// TIA Portal project "PLC_ABB_Drive" (V15)

(* hardware
DEVICE "S7-1200 station_1"  S7-1200 Station
   slot 0: "Rack_0"  S7-1200 Rack  Rack  V1.0
   slot 1: "PLC_1"  CPU 1212C DC/DC/DC  6ES7 212-1AE31-0XB0  V3.0
   slot 101: "CM 1243-5"  CM 1243-5  6GK7 243-5DX30-0XE0  V1.3
DEVICE "GSD device_1"  GSD.Device
   slot 0: "Slave_1"  6SE640X-1PB00-0AA0  V1.0
   slot 0: "Rack_0"  Rail
*)

// ===== PLC "PLC_1"  CPU 1212C DC/DC/DC =====

VAR_GLOBAL   // PLC tag table "Default tag table"
   "Tag_1" AT %ID260 : DWord;
   "Tag_2" AT %MW100 : Word;
   "InicioVariador" AT %M0.0 : Bool;
   "Tag_3" AT %M0.1 : Bool;
   "Tag_4" AT %M0.2 : Bool;
   "Tag_5" AT %M0.3 : Bool;
   "Tag_6" AT %M0.4 : Bool;
   "Tag_7" AT %M0.5 : Bool;
   "Tag_8" AT %M0.6 : Bool;
   "Tag_9" AT %M0.7 : Bool;
   "Tag_10" AT %M1.0 : Bool;
   "Tag_11" AT %M1.1 : Bool;
   "Tag_12" AT %M1.2 : Bool;
   "Tag_13" AT %M1.4 : Bool;
   "Tag_14" AT %M1.3 : Bool;
   "Tag_15" AT %M1.5 : Bool;
   "Tag_16" AT %M1.6 : Bool;
   "Tag_17" AT %M1.7 : Bool;
   "Tag_18" AT %M2.0 : Bool;
   "LeerValorParam" AT %ID260 : DWord;
   "Tag_20" AT %QW266 : Word;
   "ParametrosDeControl" AT %QW264 : Word;
   "VelocidadControl" AT %MW90 : Word;
   "ParametroControlVel." AT %QW268 : Int;
   "Tag_21" AT %IW264 : Word;
   "Parametro" AT %QW256 : Word;
   "Indice" AT %QW258 : Int;
   "Tag_24" AT %QW260 : Word;
   "ValorParametro" AT %QD260 : Real;
   "LeerParametro" AT %IW256 : Word;
   "ParamRecibido" AT %MW6 : Word;
   "LeerIndice" AT %IW258 : Int;
   "IndiceRecibido" AT %MW8 : Int;
   "VlrParamRecibido" AT %MD10 : DWord;
END_VAR

TYPE "inn"
   STRUCT
      JogDerecha : Bool;
      JogIzquierda : Bool;
      controlPLC : Bool;
      InversionGiro : Bool;
      libre : Bool;
      potenciometroarriba : Bool;
      potenciometroabajo : Bool;
      "mando-local-remoto" : Bool;
      start : Bool;
      stop : Bool;
      "stop-rapido" : Bool;
      "generador-rampa" : Bool;
      "rampa-on" : Bool;
      "rampa-off" : Bool;
      "rampa-start" : Bool;
      "alarma-fallo" : Bool;
      VelVariador : Int;
   END_STRUCT;
END_TYPE

TYPE "out1"
   STRUCT
      Setpoint_on_off : Bool;
      MasterControlReq : Bool;
      F_reached : Bool;
      Alarm_currentLim : Bool;
      MotorHoldBreake : Bool;
      MotorOverload : Bool;
      CW0_CWW1 : Bool;
      ConverterOverload : Bool;
      ReadyForOn : Bool;
      ReadyToRun : Bool;
      OperationEnable : Bool;
      Fault1 : Bool;
      Off2Command : Bool;
      Off3Command : Bool;
      StartLockout : Bool;
      Alarm : Bool;
      StatusSpeed : Int;
   END_STRUCT;
END_TYPE

DATA_BLOCK "LecturadelVariador"   // DB1
{ S7_Optimized_Access := 'FALSE' }
VERSION : 0.1
   VAR
      estadodelvariador : "out1";
   END_VAR
BEGIN
END_DATA_BLOCK

DATA_BLOCK "ControldelVariador"   // DB2
{ S7_Optimized_Access := 'FALSE' }
VERSION : 0.1
   VAR
      controlvariador : "inn";
   END_VAR
BEGIN
END_DATA_BLOCK

FUNCTION_BLOCK "Block_1"   // FB1, FBD
{ S7_Optimized_Access := 'TRUE' }
VERSION : 0.1
BEGIN
END_FUNCTION_BLOCK

ORGANIZATION_BLOCK "Main"   // OB1, LAD, ProgramCycle
TITLE = "Main Program Sweep (Cycle)"
{ S7_Optimized_Access := 'TRUE' }
VERSION : 0.1
BEGIN

REGION Network 1
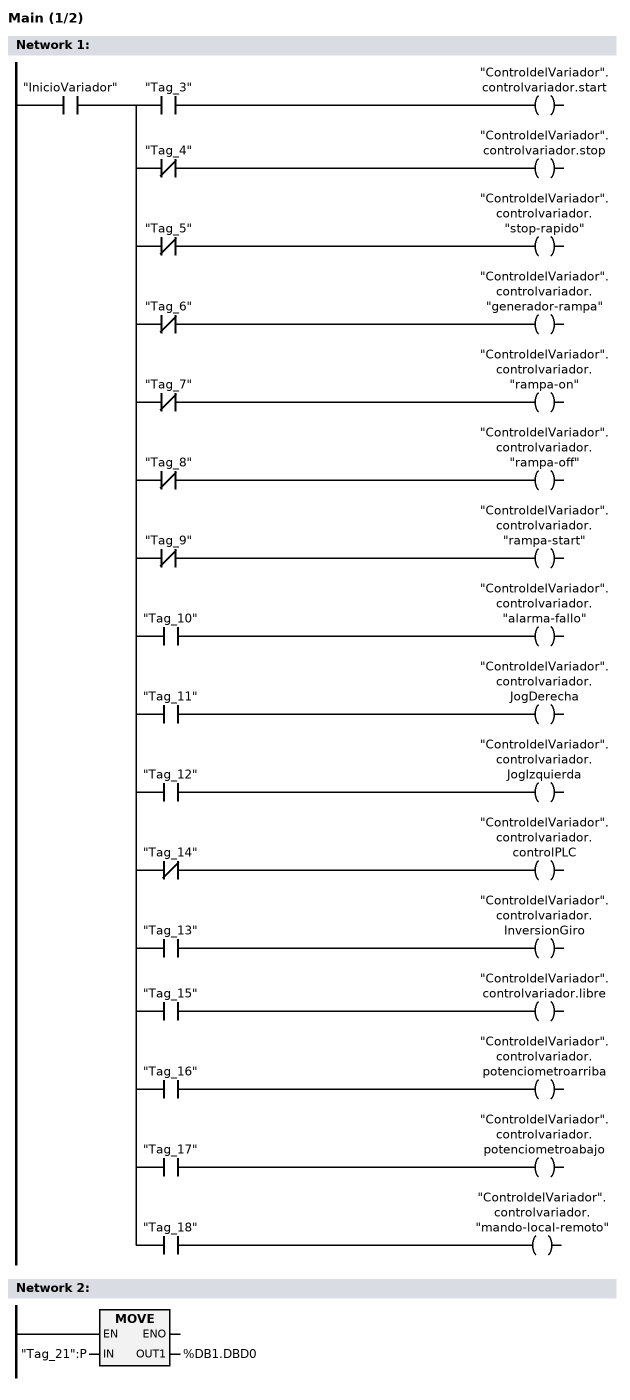
   RUNG wire#powerrail
      Contact( "InicioVariador" )
      wire#w1
      Contact( "Tag_3" )
      Coil( "ControldelVariador".controlvariador.start )
   END_RUNG
   RUNG wire#w1
      I_Contact( "Tag_4" )
      Coil( "ControldelVariador".controlvariador.stop )
   END_RUNG
   RUNG wire#w1
      I_Contact( "Tag_5" )
      Coil( "ControldelVariador".controlvariador."stop-rapido" )
   END_RUNG
   RUNG wire#w1
      I_Contact( "Tag_6" )
      Coil( "ControldelVariador".controlvariador."generador-rampa" )
   END_RUNG
   RUNG wire#w1
      I_Contact( "Tag_7" )
      Coil( "ControldelVariador".controlvariador."rampa-on" )
   END_RUNG
   RUNG wire#w1
      I_Contact( "Tag_8" )
      Coil( "ControldelVariador".controlvariador."rampa-off" )
   END_RUNG
   RUNG wire#w1
      I_Contact( "Tag_9" )
      Coil( "ControldelVariador".controlvariador."rampa-start" )
   END_RUNG
   RUNG wire#w1
      Contact( "Tag_10" )
      Coil( "ControldelVariador".controlvariador."alarma-fallo" )
   END_RUNG
   RUNG wire#w1
      Contact( "Tag_11" )
      Coil( "ControldelVariador".controlvariador.JogDerecha )
   END_RUNG
   RUNG wire#w1
      Contact( "Tag_12" )
      Coil( "ControldelVariador".controlvariador.JogIzquierda )
   END_RUNG
   RUNG wire#w1
      I_Contact( "Tag_14" )
      Coil( "ControldelVariador".controlvariador.controlPLC )
   END_RUNG
   RUNG wire#w1
      Contact( "Tag_13" )
      Coil( "ControldelVariador".controlvariador.InversionGiro )
   END_RUNG
   RUNG wire#w1
      Contact( "Tag_15" )
      Coil( "ControldelVariador".controlvariador.libre )
   END_RUNG
   RUNG wire#w1
      Contact( "Tag_16" )
      Coil( "ControldelVariador".controlvariador.potenciometroarriba )
   END_RUNG
   RUNG wire#w1
      Contact( "Tag_17" )
      Coil( "ControldelVariador".controlvariador.potenciometroabajo )
   END_RUNG
   RUNG wire#w1
      Contact( "Tag_18" )
      Coil( "ControldelVariador".controlvariador."mando-local-remoto" )
   END_RUNG
   // the same network as SCL:
   "ControldelVariador".controlvariador.start := "InicioVariador" AND "Tag_3";
   "ControldelVariador".controlvariador.stop := "InicioVariador" AND NOT "Tag_4";
   "ControldelVariador".controlvariador."stop-rapido" := "InicioVariador" AND NOT "Tag_5";
   "ControldelVariador".controlvariador."generador-rampa" := "InicioVariador" AND NOT "Tag_6";
   "ControldelVariador".controlvariador."rampa-on" := "InicioVariador" AND NOT "Tag_7";
   "ControldelVariador".controlvariador."rampa-off" := "InicioVariador" AND NOT "Tag_8";
   "ControldelVariador".controlvariador."rampa-start" := "InicioVariador" AND NOT "Tag_9";
   "ControldelVariador".controlvariador."alarma-fallo" := "InicioVariador" AND "Tag_10";
   "ControldelVariador".controlvariador.JogDerecha := "InicioVariador" AND "Tag_11";
   "ControldelVariador".controlvariador.JogIzquierda := "InicioVariador" AND "Tag_12";
   "ControldelVariador".controlvariador.controlPLC := "InicioVariador" AND NOT "Tag_14";
   "ControldelVariador".controlvariador.InversionGiro := "InicioVariador" AND "Tag_13";
   "ControldelVariador".controlvariador.libre := "InicioVariador" AND "Tag_15";
   "ControldelVariador".controlvariador.potenciometroarriba := "InicioVariador" AND "Tag_16";
   "ControldelVariador".controlvariador.potenciometroabajo := "InicioVariador" AND "Tag_17";
   "ControldelVariador".controlvariador."mando-local-remoto" := "InicioVariador" AND "Tag_18";
END_REGION

REGION Network 2
   RUNG wire#powerrail
      { S7_GenerateENO := "TRUE" } Move(in := "Tag_21":P, out1 => %DB1.DBD0)
   END_RUNG
   // the same network as SCL:
   %DB1.DBD0 := "Tag_21":P;
END_REGION

REGION Network 3
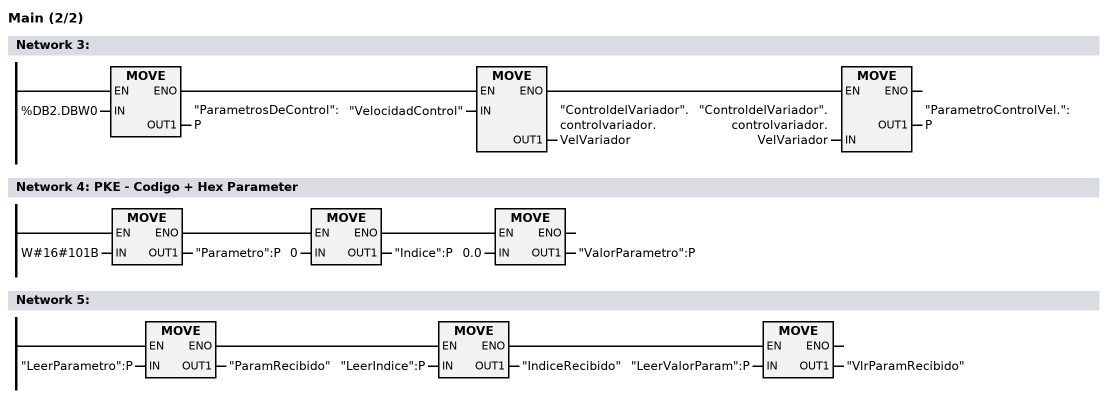
   RUNG wire#powerrail
      { S7_GenerateENO := "TRUE" } Move(in := %DB2.DBW0, out1 => "ParametrosDeControl":P)
      { S7_GenerateENO := "TRUE" } Move(in := "VelocidadControl", out1 => "ControldelVariador".controlvariador.VelVariador)
      { S7_GenerateENO := "TRUE" } Move(in := "ControldelVariador".controlvariador.VelVariador, out1 => "ParametroControlVel.":P)
   END_RUNG
   // the same network as SCL:
   // ENO of a box is taken as its EN; it also drops when the box reports an error
   "ParametrosDeControl":P := %DB2.DBW0;
   "ControldelVariador".controlvariador.VelVariador := "VelocidadControl";
   "ParametroControlVel.":P := "ControldelVariador".controlvariador.VelVariador;
END_REGION

REGION Network 4: PKE - Codigo + Hex Parameter
   RUNG wire#powerrail
      { S7_GenerateENO := "TRUE" } Move(in := W#16#101B, out1 => "Parametro":P)
      { S7_GenerateENO := "TRUE" } Move(in := 0, out1 => "Indice":P)
      { S7_GenerateENO := "TRUE" } Move(in := 0.0, out1 => "ValorParametro":P)
   END_RUNG
   // the same network as SCL:
   // ENO of a box is taken as its EN; it also drops when the box reports an error
   "Parametro":P := W#16#101B;
   "Indice":P := 0;
   "ValorParametro":P := 0.0;
END_REGION

REGION Network 5
   RUNG wire#powerrail
      { S7_GenerateENO := "TRUE" } Move(in := "LeerParametro":P, out1 => "ParamRecibido")
      { S7_GenerateENO := "TRUE" } Move(in := "LeerIndice":P, out1 => "IndiceRecibido")
      { S7_GenerateENO := "TRUE" } Move(in := "LeerValorParam":P, out1 => "VlrParamRecibido")
   END_RUNG
   // the same network as SCL:
   // ENO of a box is taken as its EN; it also drops when the box reports an error
   "ParamRecibido" := "LeerParametro":P;
   "IndiceRecibido" := "LeerIndice":P;
   "VlrParamRecibido" := "LeerValorParam":P;
END_REGION
END_ORGANIZATION_BLOCK